(* PLC project poST.project, poSTIDE *)
(* stored: creationDateTime 2021-08-31T00:00:00.000000 *)

FUNCTION ADD_DT_TIME : DATE_AND_TIME
  VAR_INPUT
    in1 : DATE_AND_TIME;
    in2 : TIME;
  END_VAR

END_FUNCTION
